// TIA Portal V20 export
DATA_BLOCK "BK11"   // DB305
// stored: MemoryReserve 100
   VAR
      "X10-1.ANODE NG BOX FULL SENSOR" : Bool := TRUE;
      "X10-2.SPARE" : Bool := FALSE;
      "X12-1.ANODE NG BOX LIFT DOWN" : Bool := FALSE;
      "X12-2.ANODE NG BOX LIFT UP" : Bool := TRUE;
      "X14-1.ANODE NG BOX LOCK DOWN" : Bool := TRUE;
      "X14-2.ANODE NG BOX LOCK UP" : Bool := FALSE;
      "X16-1.ANODE NG BOX NG BOX DETECT SENSOR" : Bool := TRUE;
      "X16-2.SPARE" : Bool := FALSE;
   END_VAR
BEGIN
END_DATA_BLOCK
